// TwinCAT 3 PLC project PlcHammer
// Title: PlcHammer
// Company: Vortex.Library
// ProjectVersion: 0.6.0.913
// ProgramVersion: 3.1.4023.0
// libraries:
//   Tc2_Math, * (Beckhoff Automation GmbH)
//   Tc2_Standard, * (Beckhoff Automation GmbH)
//   Tc2_System, * (Beckhoff Automation GmbH)
//   Tc3_Module, * (Beckhoff Automation GmbH)
//   TcoCore, 0.6.0.913 (Vortex.Library)
//   TcoData, 0.6.0.913 (Vortex.Library)
//   TcoDrivesBeckhoff, 0.6.0.913 (Vortex.Library)
//   TcoElements, 0.6.0.913 (Vortex.Library)
//   TcoInspectors, 0.6.0.913 (Vortex.Library)
//   TcoIo, 0.6.0.913 (Vortex.Library)
//   TcoPneumatics, 0.6.0.913 (Vortex.Library)
//   TcoUtilities, 0.6.0.913 (Vortex.Library)
// project tree:
//   Components/Drive/ DriveSim.TcPOU, DriveSimMoveAbsoluteTask.TcPOU, IDrive.TcIO
//   DUTs/ enumModes.TcDUT
//   Misc/Checkers/ Checkers.TcPOU, AnalogueValueCheck.TcDUT, eCheckResult.TcDUT
//   / PlcTask.TcTTO
//   POUs/ AppContext.TcPOU, TECH_MAIN.TcPOU
//   POUs/Data/ ProcessDataManager.TcPOU, RealValueSimulation.TcPOU, TechnologicalDataManager.TcPOU
//   POUs/Station001/ Station001_Swift.TcPOU, IO.TcGVL, Station001.TcPOU, Station001_Components.TcPOU, Station001_GroundMode.TcPOU, Station001_AutomatMode.TcPOU, Station001_ProductionData.TcDUT, Station001_TechnologicalSettings.TcDUT
// real-time tasks:
//   TASK PlcTask: cycle T#10ms, priority 20, ADS port 350
// motion (NC):
//   TASK NC-Task 1 SAF: cycle T#2ms, priority 4, ADS port 501
//   TASK NC-Task 1 SVB: cycle T#10ms, priority 8, ADS port 511
//   AXIS Axis 1 (id 1)
//     OtherSettings: AllowMotionCmdToSlave=true
//     encoder EncType=1
//     drive DrvType=5
//       Analog: TorqueSetpointScale=10, ScaleFactorActTorque=0.1
//       TimeComp: TaskDelayCycles=1
//     controller CtrType=1
//       CtrPara: PriorControlFactor=1
//         Observer: BandWidth=20
// variable links:
//   PlcHammer/PlcHammer Instance <-> NC-Task 1 SAF/Axes/Axis 1
//     PlcTask Inputs/IO.Axis1.NcToPlc <-> Outputs/ToPlc
//     PlcTask Outputs/IO.Axis1.PlcToNc <-> Inputs/FromPlc

CONFIGURATION PlcHammer
    RESOURCE PLC ON TwinCAT3
        TASK PlcTask(INTERVAL := T#10ms, PRIORITY := 20);
        PROGRAM TECH_MAIN WITH PlcTask : TECH_MAIN;
    END_RESOURCE
END_CONFIGURATION

// ---- DUTs/enumModes.TcDUT
{attribute 'qualified_only'}
{attribute 'strict'}
TYPE enumModes :
(
    Idle := 0,
    Automat := 1000,
    Ground := 2000,
    Service := 3000
);
END_TYPE

// ---- Misc/Checkers/AnalogueValueCheck.TcDUT
{attribute wpf [Container(Layout.Wrap)]}
{attribute wpf [Group(Layout.GroupBox)]}
TYPE AnalogueValueCheck :
STRUCT
    Mininum : REAL;
    {attribute clr [RenderIgnore("ShadowControl", "ShadowControlSlim")]}
    Measured : REAL;
    Maximum : REAL;
END_STRUCT
END_TYPE

// ---- Misc/Checkers/eCheckResult.TcDUT
{attribute 'qualified_only'}
{attribute 'strict'}
TYPE eCheckResult :
(
    None := 0,
    Passed := 10,
    Failed := 20
);
END_TYPE

// ---- POUs/Station001/Station001_ProductionData.TcDUT
TYPE Station001_ProductionData EXTENDS TcoData.TcoEntity :
STRUCT
    {attribute clr [Container(Layout.Stack)]}
    Result : TcoComprehensiveResult;
    RecipeName : STRING;
    DimX : TcoInspectors.TcoAnalogueInspector(THISSTRUCT);
    DimY : TcoInspectors.TcoAnalogueInspector(THISSTRUCT);
    DimZ : TcoInspectors.TcoAnalogueInspector(THISSTRUCT);
END_STRUCT
END_TYPE

// ---- POUs/Station001/Station001_TechnologicalSettings.TcDUT
TYPE Station001_TechnologicalSettings EXTENDS TcoData.TcoEntity :
STRUCT
    LoadPartsHorizontalPosition : LREAL;
    PassedPartsHorizontalPosition : LREAL;
    FailedPartsHorizontalPosition : LREAL;
    AxisSpeed : LREAL;
    AxisAcc : LREAL;
    AxisDcc : LREAL;
    AxisJerk : LREAL;
END_STRUCT
END_TYPE

// ---- POUs/Station001/IO.TcGVL
{attribute 'qualified_only'}
VAR_GLOBAL
    iA1 AT %I* : ARRAY[0..7] OF BOOL;
    iA2 AT %I* : ARRAY[0..7] OF BOOL;
    qA1 AT %Q* : ARRAY[0..7] OF BOOL;
    qA2 AT %Q* : ARRAY[0..7] OF BOOL;
    Axis1 : TcoDrivesBeckhoff.TcoAxisRef;
END_VAR

// ---- Components/Drive/IDrive.TcIO
INTERFACE IDrive

METHOD MoveAbsolute : TcoCore.ITcoTaskStatus
VAR_INPUT
	TargetPosition : LREAL;
END_VAR
END_METHOD

PROPERTY MoveAbsoluteTask : REFERENCE TO DriveSimMoveAbsoluteTask
GET
END_GET
END_PROPERTY

END_INTERFACE

// ---- POUs/TECH_MAIN.TcPOU
PROGRAM TECH_MAIN
VAR
    _app : AppContext;
END_VAR

_app.Run();
_app.RtcSynchronize(TRUE, '', 60);

END_PROGRAM

// ---- POUs/AppContext.TcPOU
FUNCTION_BLOCK AppContext EXTENDS TcoCore.TcoContext
VAR
    _station001 : Station001(THIS^);
END_VAR

(*~
    <docu>
        <summary>
            Main method of the TcoContext. This is the entry point of any control logic that belongs to this context.
            The call of this method is ensured by calling the <c>InstanceName.Run()</c> method, and it must not be called explicitly.
            This method is abstract, and it must be overridden in derived block.
        </summary>
    </docu>
~*)
METHOD PROTECTED Main
THIS^.RtcSynchronize(TRUE, '', 60);
_station001();
END_METHOD

END_FUNCTION_BLOCK

// ---- POUs/Station001/Station001.TcPOU
FUNCTION_BLOCK Station001 EXTENDS TcoCore.TcoObject
VAR
    _components : Station001_Components(THIS^);
    _groundMode : Station001_GroundMode(THIS^, eRestoreMode.None);
    _automatMode : Station001_AutomatMode(THIS^, eRestoreMode.None);
    _swiftSequence : Station001_Swift(THIS^, eRestoreMode.None);
    _groundModeTask : TcoCore.TcoTask(THIS^);
    _automatModeTask : TcoCore.TcoTask(THIS^);
    _serviceModeTask : TcoCore.TcoTask(THIS^);
    _swiftModeTask : TcoCore.TcoTask(THIS^);
    _processRecipies : ProcessDataManager(THIS^);
    _processTraceabilty : ProcessDataManager(THIS^);
    _technologicalDataManager : TechnologicalDataManager(THIS^);
    _currentMode : enumModes := enumModes.Idle;
    _checkers : Checkers(THIS^);
    _externalToken : STRING;
    _externalTokenPresence : BOOL;
END_VAR

_components();
_processRecipies();
_processTraceabilty();
_technologicalDataManager();
ServiceMode();
GroundMode();
AutomatMode();

IF (_swiftModeTask.Execute()) THEN
    Messenger.Trace('Service mode active');
    _automatModeTask.Restore();
    _groundModeTask.Restore();
    _groundMode.Restore();
    _automatMode.Restore();
    _serviceModeTask.Restore();
    _swiftSequence.Run();
    _currentMode := enumModes.Idle;
END_IF

METHOD AutomatMode : BOOL
VAR_INPUT
END_VAR
_automatModeTask.Enabled := _groundModeTask.Done;

IF (_automatModeTask.Execute()) THEN
    Messenger.Trace('Automat mode active');
    _serviceModeTask.Abort();
    _automatMode.Run();
    _currentMode := enumModes.Automat;
END_IF
END_METHOD

PROPERTY Checkers : REFERENCE TO Checkers
GET
Checkers REF= _checkers;
END_GET
END_PROPERTY

PROPERTY Components : REFERENCE TO Station001_Components
GET
Components REF= _components;
END_GET
END_PROPERTY

METHOD GroundMode : BOOL
VAR_INPUT
END_VAR
IF (_groundModeTask.Execute()) THEN
    Messenger.Trace('Ground position mode active');
    _serviceModeTask.Restore();
    _automatModeTask.Restore();
    _automatMode.Restore();
    _groundMode.Run();
    _groundModeTask.DoneWhen(_groundMode.CurrentStep.ID = 300);

    IF _groundModeTask.Done THEN
        _groundMode.Restore();
    END_IF

    _currentMode := enumModes.Ground;
END_IF
END_METHOD

PROPERTY ProcessRecepie : REFERENCE TO ProcessDataManager
GET
ProcessRecepie REF= _processRecipies;
END_GET
END_PROPERTY

PROPERTY ProcessTraceabilty : REFERENCE TO ProcessDataManager
GET
ProcessTraceabilty REF= _processTraceabilty;
END_GET
END_PROPERTY

PROPERTY ProductionData : REFERENCE TO Station001_ProductionData
GET
ProductionData REF= _processTraceabilty._data;
END_GET
END_PROPERTY

METHOD ServiceMode
VAR_INPUT
END_VAR
IF (_serviceModeTask.Execute()) THEN
    Messenger.Trace('Service mode active');
    _automatModeTask.Restore();
    _groundModeTask.Restore();
    _groundMode.Restore();
    _automatMode.Restore();
    _components.Service();
    _currentMode := enumModes.Service;
END_IF
END_METHOD

PROPERTY TechnologicalDataManager : REFERENCE TO TechnologicalDataManager
GET
TechnologicalDataManager REF= _technologicalDataManager;
END_GET
END_PROPERTY

END_FUNCTION_BLOCK

// ---- POUs/Station001/Station001_Components.TcPOU
{attribute wpf [Container(Layout.Stack)]}
FUNCTION_BLOCK Station001_Components EXTENDS TcoCore.TcoObject
VAR
    //	_horizontalAxis : DriveSim(THIS^);
    {attribute addProperty Name "Horizontal axis"}
    _horizontalNcAxis : TcoDrivesBeckhoff.TcoDriveSimple(THIS^);
    {attribute addProperty Name "Vertical piston"}
    {attribute addProperty _moveHomeDefaultName "<#MOVE HOME#>"}
    {attribute addProperty _moveWorkDefaultName "<#MOVE TO WORK#>"}
    {attribute addProperty _stopDefaultName "<#STOP#>"}
    _verticalPiston : TcoPneumatics.TcoCylinder(THIS^);
    {attribute addProperty Name "Gripper piston"}
    {attribute addProperty _moveHomeDefaultName "<#MOVE HOME#>"}
    {attribute addProperty _moveWorkDefaultName "<#MOVE TO WORK#>"}
    {attribute addProperty _stopDefaultName "<#STOP#>"}
    _gripperPiston : TcoPneumatics.TcoCylinder(THIS^);
END_VAR
(* Simulation variables *)
VAR
    _counterSimVerticalPiston : ULINT;
    _counterSimGripperPiston : ULINT;
    _simulationCycleVerticalPiston : BOOL;
    _simulationCycleGripperPiston : BOOL;
    _verticalPosition : INT;
    _gripperPosition : INT;
    _dimXsim : RealValueSimulation;
    _dimYsim : RealValueSimulation;
    _dimZsim : RealValueSimulation;
    _dimX : REAL;
    _dimY : REAL;
    _dimZ : REAL;
END_VAR
VAR CONSTANT
    _verticalPistonStroke : INT := 150;
    _gripperPistonStroke : INT := 50;
END_VAR

Simulation();

_verticalPiston(inoAtHomePos := IO.iA1[0],
    inoAtWorkPos := IO.iA1[1],
    inoToHomePos := IO.qA1[0],
    inoToWorkPos := IO.qA1[1]);

_gripperPiston(inoAtHomePos := IO.iA1[2],
    inoAtWorkPos := IO.iA1[3],
    inoToHomePos := IO.qA1[2],
    inoToWorkPos := IO.qA1[3]);

//_horizontalAxis();
_horizontalNcAxis(inEnable := TRUE,
    inEnablePositive := TRUE,
    inEnableNegative := TRUE,
    inCalibrationCam := FALSE,
    inoAxisRef := IO.Axis1);

PROPERTY Gripper : REFERENCE TO TcoPneumatics.TcoCylinder
GET
Gripper REF= _gripperPiston;
END_GET
END_PROPERTY

PROPERTY HorizontalNcAxis : TcoDrivesBeckhoff.ITcoDriveSimple
GET
HorizontalNcAxis := _horizontalNcAxis;
END_GET
END_PROPERTY

METHOD Service : BOOL
VAR_INPUT
END_VAR
//_horizontalAxis.Service();
_horizontalNcAxis.Service();
_verticalPiston.Service();
_gripperPiston.Service();
END_METHOD

METHOD Simulation
VAR_INPUT
END_VAR
IF (_verticalPiston.MoveHomeTask.Busy OR _verticalPiston.MoveWorkTask.Busy) THEN
    _counterSimVerticalPiston := _counterSimVerticalPiston + 1;
    _simulationCycleVerticalPiston := (_counterSimVerticalPiston MOD _verticalPistonStroke) = 0;
END_IF;

IF (Gripper.MoveHomeTask.Busy OR Gripper.MoveWorkTask.Busy) THEN
    _counterSimGripperPiston := _counterSimVerticalPiston + 1;
    _simulationCycleGripperPiston := (_counterSimVerticalPiston MOD _gripperPistonStroke) = 0;
END_IF;

IF (IO.qA1[0] AND _simulationCycleVerticalPiston) THEN
    IO.iA1[0] := TRUE;
    IO.iA1[1] := FALSE;
    _verticalPosition := 0;
END_IF

IF (IO.qA1[1] AND _simulationCycleVerticalPiston) THEN
    IO.iA1[1] := TRUE;
    IO.iA1[0] := FALSE;
    _verticalPosition := _verticalPistonStroke;
END_IF

IF (IO.qA1[0] AND NOT IO.iA1[0]) THEN
    _verticalPosition := (_verticalPosition - 1);
END_IF;

IF (IO.qA1[1] AND NOT IO.iA1[1]) THEN
    _verticalPosition := (_verticalPosition + 1);
END_IF;

IF (IO.qA1[2] AND _simulationCycleVerticalPiston) THEN
    IO.iA1[2] := TRUE;
    IO.iA1[3] := FALSE;
    _gripperPosition := 0;
END_IF

IF (IO.qA1[3] AND _simulationCycleVerticalPiston) THEN
    IO.iA1[3] := TRUE;
    IO.iA1[2] := FALSE;
    _gripperPosition := _gripperPistonStroke;
END_IF

IF (IO.qA1[2] AND NOT IO.iA1[2]) THEN
    _gripperPosition := (_gripperPosition - 1);
END_IF;

IF (IO.qA1[3] AND NOT IO.iA1[3]) THEN
    _gripperPosition := (_gripperPosition + 1);
END_IF

_dimXsim.Dc := 3;
_dimYsim.Dc := 3;
_dimZsim.Dc := 3;
_dimXsim.P1 := 0.74;
_dimYsim.P1 := 0.74;
_dimZsim.P1 := 0.74;
_dimXsim.P2 := 1.1;
_dimYsim.P2 := 1.1;
_dimZsim.P2 := 1.1;
END_METHOD

PROPERTY VerticalAxis : REFERENCE TO TcoPneumatics.TcoCylinder
GET
VerticalAxis REF= _verticalPiston;
END_GET
END_PROPERTY

END_FUNCTION_BLOCK

// ---- POUs/Data/RealValueSimulation.TcPOU
FUNCTION_BLOCK RealValueSimulation
VAR_INPUT
    inMinValue : REAL;
    inMaxValue : REAL;
END_VAR
VAR_IN_OUT
    inoutValue : REAL;
END_VAR
VAR
    _dc : LREAL := 5.4;
    _min : REAL;
    _max : REAL;
    _p1 : LREAL := 2;
    _p2 : LREAL := 3.5;
    _x0 : LREAL;
    _x1 : LREAL;
    _pm : LREAL;
    _ex : LREAL;
END_VAR

_ex := EXPT(10, _dc);
_x0 := inoutValue * _ex;

IF _x0 = 0 THEN
    _x0 := (inMaxValue + inMinValue) / 2 * _ex;
END_IF

_min := inMinValue * _ex;
_max := inMaxValue * _ex;
_pm := (_max - _min);
_x1 := _min + (Tc2_Math.LMOD((_x0 * _p1 + _p2), _pm));
inoutValue := Tc2_Math.LTRUNC(_x1 / _ex);

PROPERTY Dc : LREAL
GET
Dc := _dc;
END_GET
SET
_dc := Dc;
END_SET
END_PROPERTY

PROPERTY P1 : LREAL
GET
P1 := _p1;
END_GET
SET
_p1 := P1;
END_SET
END_PROPERTY

PROPERTY P2 : LREAL
GET
P2 := _p2;
END_GET
SET
_p2 := P2;
END_SET
END_PROPERTY

END_FUNCTION_BLOCK

// ---- POUs/Station001/Station001_GroundMode.TcPOU
FUNCTION_BLOCK Station001_GroundMode EXTENDS TcoCore.TcoSequencer

(*~
    <docu>
        <summary>
            Main method of the sequener. Custom code needs to be placed here. The sequencer is executed by call of InstanceName.Run() method.
            This method is abstract, and it must be overridden in derived block.
        </summary>
    </docu>
~*)
METHOD PROTECTED Main : BOOL
VAR CONSTANT
    HORIZONTAL_AXIS_HOME_POSITION : LREAL := 0.0;
END_VAR
IF (Step(10, TRUE, 'RESTORE ALL COMPONENTS')) THEN
    //--------------------------------------------
    Station.Components._horizontalNcAxis.Restore();
    Station.Components._verticalPiston.Restore();
    Station.Components._gripperPiston.Restore();
    StepCompleteWhen(TRUE);
    //--------------------------------------------
END_IF;

IF (Step(100, TRUE, 'MOVE VERTICAL AXIS UP')) THEN
    //--------------------------------------------
    StepCompleteWhen(Station.Components.VerticalAxis.MoveToHome().Done);
    //--------------------------------------------
END_IF;

IF (Step(125, TRUE, 'LOAD TECHNOLOGICAL SETTINGS')) THEN
    //--------------------------------------------
    StepCompleteWhen(Station.TechnologicalDataManager.Read('default').Done);
    //--------------------------------------------
END_IF;

IF (Step(150, NOT Station.Components.HorizontalNcAxis.DriveRef._axisStatus.Homed, 'HORIZONTAL AXIS HOMING')) THEN
    //--------------------------------------------
    StepCompleteWhen(Station.Components.HorizontalNcAxis.DriveRef.Home(inPosition := 0,
            inHomingMode := TcoDrivesBeckhoff.eHomingMode.MC_Direct,
            inClearPositionLag := FALSE,
            inSearchDirection := TcoDrivesBeckhoff.eDirection.MC_Undefined_Direction,
            inSearchVelocity := 100.0,
            inSyncDirection := TcoDrivesBeckhoff.eDirection.MC_Undefined_Direction,
            inSyncVelocity := 100.0,
            inReferenceMode := TcoDrivesBeckhoff.eEncoderReferenceMode.ENCODERREFERENCEMODE_DEFAULT).Done);
    //--------------------------------------------
END_IF;

IF (Step(200, TRUE, 'MOVE HORIZONTAL AXIS TO BASE POSITION & OPEN GRIPPER')) THEN
    //--------------------------------------------
    IF (Station.Components.HorizontalNcAxis.DriveRef.MoveAbsolute(HORIZONTAL_AXIS_HOME_POSITION,
        THIS^.Station.TechnologicalDataManager._data.AxisSpeed,
        THIS^.Station.TechnologicalDataManager._data.AxisAcc,
        THIS^.Station.TechnologicalDataManager._data.AxisDcc,
        THIS^.Station.TechnologicalDataManager._data.AxisJerk).Done AND
        Station.Components.Gripper.MoveToHome().Done) THEN
        CompleteStep();
    END_IF;
    //--------------------------------------------
END_IF;

IF (Step(300, TRUE, 'GROUND POSITION DONE')) THEN
    //--------------------------------------------
    ;
    //--------------------------------------------
END_IF;
END_METHOD

(*~
    <docu>
        <summary>
            This method is executed upon step completion.
            This method can be overridden in derived block by custom logic.
        </summary>
    </docu>
~*)
METHOD PROTECTED OnStepCompleted
END_METHOD

PROPERTY Station : REFERENCE TO Station001
GET
VAR
    _station : POINTER TO Station001;
END_VAR
IF __QUERYPOINTER(Parent, _station) THEN // Check if _Parent is Station001
    Station REF= _station^; // If the check is successful dereference a pointer. simlar to THIS^ or SUPER^
END_IF
END_GET
END_PROPERTY

END_FUNCTION_BLOCK

// ---- POUs/Data/TechnologicalDataManager.TcPOU
FUNCTION_BLOCK TechnologicalDataManager EXTENDS TcoData.TcoDataExchange
VAR
    //this variable has to called "_data" - PC app will access this variable by its name.
    _data : Station001_TechnologicalSettings := (Parent := THIS^);
END_VAR

SUPER^();
//Set som default values in case of no setting loaded to the PLC yet.
//IF _data.LoadPartsHorizontalPosition = 0  AND _data.FailedPartsHorizontalPosition = 0 AND _data.PassedPartsHorizontalPosition = 0 THEN
//    _data.LoadPartsHorizontalPosition := 50;
//    _data.FailedPartsHorizontalPosition := 300.0;
//    _data.PassedPartsHorizontalPosition := 450.0;
//END_IF
//IF _data.AxisSpeed = 0 THEN
//    _data.AxisSpeed := 1000.0;
//END_IF
//IF _data.AxisAcc = 0 THEN
//    _data.AxisAcc := 10000.0;
//END_IF
//IF _data.AxisDcc = 0 THEN
//    _data.AxisDcc := 10000.0;
//END_IF
//IF _data.AxisJerk = 0 THEN
//    _data.AxisJerk := 50000.0;
//END_IF

END_FUNCTION_BLOCK

// ---- POUs/Station001/Station001_AutomatMode.TcPOU
FUNCTION_BLOCK Station001_AutomatMode EXTENDS TcoCore.TcoSequencer
VAR
    _partPassedChecks : BOOL;
    _groupInspection : TcoInspectors.TcoInspectionGroup(THIS^);
    _dialog : TcoCore.TcoDialog(THIS^);
END_VAR

(*~
    <docu>
        <summary>
            Main method of the sequener. Custom code needs to be placed here. The sequencer is executed by call of InstanceName.Run() method.
            This method is abstract, and it must be overridden in derived block.
        </summary>
    </docu>
~*)
METHOD PROTECTED Main : BOOL
VAR CONSTANT
    HORIZONTAL_AXIS_HOME_POSITION : LREAL := 100.0;
END_VAR
VAR_INST
    _id : STRING;
END_VAR
IF (Step(0, TRUE, 'DIALOG - DO WE CONTINUE')) THEN
    //--------------------------------------------
    IF (_dialog.Show().WithOk().WithCaption('What`s next?').WithText('To continue click OK?').Answer = TcoCore.eDialogAnswer.OK) THEN
        CompleteStep();
    END_IF;
    //--------------------------------------------
END_IF;

IF (Step(10, TRUE, 'MOVE HORIZONTAL TO LOAD')) THEN
    //--------------------------------------------
    StepCompleteWhen(Station.Components.HorizontalNCAxis.DriveRef
            .MoveAbsolute(THIS^.Station.TechnologicalDataManager._data.LoadPartsHorizontalPosition,
                THIS^.Station.TechnologicalDataManager._data.AxisSpeed,
                THIS^.Station.TechnologicalDataManager._data.AxisAcc,
                THIS^.Station.TechnologicalDataManager._data.AxisDcc,
                THIS^.Station.TechnologicalDataManager._data.AxisJerk).Done);
    //--------------------------------------------
END_IF;

IF (Step(25, TRUE, 'LOAD TECHNOLOGICAL SETTINGS')) THEN
    //--------------------------------------------
    IF (NOT Station.TechnologicalDataManager.Messenger.OnCondition(Station.TechnologicalDataManager._data._EntityId = '')
        .Error('Technological settings not selected.')
        .Pin().Pinned) THEN
        ;
        StepCompleteWhen(Station.TechnologicalDataManager.Read(Identifier := Station.TechnologicalDataManager._data._EntityId).Done);
    END_IF;
    //--------------------------------------------
END_IF;

IF (Step(50, TRUE, 'LOAD RECIPE SETTINGS')) THEN
    //--------------------------------------------
    IF (NOT Station.ProcessRecepie.Messenger.OnCondition(Station.ProcessRecepie._data._EntityId = '').Error('Process settings not selected.').Pin()
        .Pinned) THEN
        StepCompleteWhen(Station.ProcessRecepie.Read(Identifier := Station.ProcessRecepie._data._EntityId).Done);
        Station.ProductionData := Station.ProcessRecepie._data;
    END_IF

    //--------------------------------------------
END_IF;

IF (Step(100, TRUE, 'MOVE VERTICAL AXIS DOWN')) THEN
    //--------------------------------------------
    StepCompleteWhen(Station.Components.VerticalAxis.MoveToWork().Done);
    //--------------------------------------------
END_IF;

IF (Step(150, TRUE, 'GENERATE SIMULATED VALUES')) THEN
    //--------------------------------------------
    Station.Components._dimXsim(inMinValue := Station.ProductionData.DimX.Data.RequiredMin + 50,
        inMaxValue := Station.ProductionData.DimX.Data.RequiredMax - 50,
        inoutValue := Station.Components._dimX);

    Station.Components._dimYsim(inMinValue := Station.ProductionData.DimY.Data.RequiredMin + 50,
        inMaxValue := Station.ProductionData.DimY.Data.RequiredMax - 50,
        inoutValue := Station.Components._dimY);

    Station.Components._dimZsim(inMinValue := Station.ProductionData.DimZ.Data.RequiredMin + 50,
        inMaxValue := Station.ProductionData.DimZ.Data.RequiredMax - 50,
        inoutValue := Station.Components._dimZ);

    StepCompleteWhen(TRUE);
    //--------------------------------------------
END_IF;

IF (Step(200, TRUE, 'CHECK DIMENSIONS')) THEN
    //--------------------------------------------
    _groupInspection.WithCoordinator(THIS^)
        .Act()
        .Inspect(Station.ProcessTraceabilty._data.DimX.Inspect(Station.Components._dimX))
        .Inspect(Station.ProcessTraceabilty._data.DimY.Inspect(Station.Components._dimY))
        .Inspect(Station.ProcessTraceabilty._data.DimZ.Inspect(Station.Components._dimZ))
        .UpdateComprehensiveResult(Station.ProcessTraceabilty._data.Result)
        .OnFail().Dialog(200);
    //--------------------------------------------
END_IF;

IF (Step(300, TRUE, 'CLOSE GRIPPER')) THEN
    //--------------------------------------------
    StepCompleteWhen(Station.Components.Gripper.MoveToWork().Done);
    //--------------------------------------------
END_IF;

IF (Step(400, TRUE, 'MOVE VERTICAL AXIS UP')) THEN
    //--------------------------------------------
    StepCompleteWhen(Station.Components.VerticalAxis.MoveToHome().Done);
    //--------------------------------------------
END_IF;

IF (Step(425, _partPassedChecks, 'MOVE HORIZONTAL AXIS TO UNLOAD POSITION (PASSED CONVEYOR)')) THEN
    //--------------------------------------------
    StepCompleteWhen(Station.Components.HorizontalNcAxis.DriveRef
            .MoveAbsolute(THIS^.Station.TechnologicalDataManager._data.PassedPartsHorizontalPosition,
                THIS^.Station.TechnologicalDataManager._data.AxisSpeed,
                THIS^.Station.TechnologicalDataManager._data.AxisAcc,
                THIS^.Station.TechnologicalDataManager._data.AxisDcc,
                THIS^.Station.TechnologicalDataManager._data.AxisJerk).Done);
    //--------------------------------------------
END_IF;

IF (Step(450, NOT _partPassedChecks, 'MOVE HORIZONTAL AXIS TO UNLOAD POSITION (FAILED CONVEYOR)')) THEN
    //--------------------------------------------
    StepCompleteWhen(Station.Components.HorizontalNcAxis.DriveRef
            .MoveAbsolute(THIS^.Station.TechnologicalDataManager._data.FailedPartsHorizontalPosition,
                THIS^.Station.TechnologicalDataManager._data.AxisSpeed,
                THIS^.Station.TechnologicalDataManager._data.AxisAcc,
                THIS^.Station.TechnologicalDataManager._data.AxisDcc,
                THIS^.Station.TechnologicalDataManager._data.AxisJerk).Done);
    //--------------------------------------------
END_IF;

IF (Step(500, TRUE, 'MOVE VERTICAL AXIS TO UNLOAD POSITION')) THEN
    //--------------------------------------------
    StepCompleteWhen(Station.Components.VerticalAxis.MoveToWork().Done);
    //--------------------------------------------
END_IF;

IF (Step(600, TRUE, 'OPEN GRIPPER')) THEN
    //--------------------------------------------
    StepCompleteWhen(Station.Components.Gripper.MoveToHome().Done);
    //--------------------------------------------
END_IF;

IF (Step(700, TRUE, 'MOVE VERTICAL UP')) THEN
    //--------------------------------------------
    StepCompleteWhen(Station.Components.VerticalAxis.MoveToHome().Done);
    //--------------------------------------------
END_IF;

IF (Step(800, TRUE, 'MOVE HORIZONTAL TO LOAD - ASYNC')) THEN
    //--------------------------------------------
    Station.Components.HorizontalNCAxis.DriveRef.MoveAbsolute(THIS^.Station.TechnologicalDataManager._data.LoadPartsHorizontalPosition,
        THIS^.Station.TechnologicalDataManager._data.AxisSpeed,
        THIS^.Station.TechnologicalDataManager._data.AxisAcc,
        THIS^.Station.TechnologicalDataManager._data.AxisDcc,
        THIS^.Station.TechnologicalDataManager._data.AxisJerk);

    StepCompleteWhen(TRUE);
    //--------------------------------------------
END_IF;

IF (Step(840, TRUE, 'CHECK THAT THE HORIZONTAL AXIS IS IN POSITION')) THEN
    //--------------------------------------------
    _id := ULINT_TO_STRING(THIS^.Context.RealTimeClock.TickClock());
    StepCompleteWhen(TRUE);
    //--------------------------------------------
END_IF;

IF (Step(850, TRUE, 'SAVE DATA')) THEN
    //--------------------------------------------
    StepCompleteWhen(Station.ProcessTraceabilty.Create(Identifier := _id).Done);
    //--------------------------------------------
END_IF;

IF (Step(900, TRUE, 'CHECK THAT THE HORIZONTAL AXIS IS IN POSITION')) THEN
    //--------------------------------------------
    StepCompleteWhen(Station.Components.HorizontalNcAxis.DriveRef.MoveAbsoluteTask.Done);
    //--------------------------------------------
END_IF;

IF (Step(THIS^.RESTORE_STEP_ID, TRUE, 'MOVE VERTICAL AXIS UP')) THEN
    //--------------------------------------------
    StepCompleteWhen(Station.Components.VerticalAxis.MoveToHome().Done);
    //--------------------------------------------
END_IF;

IF (Step(37000, TRUE, 'MOVE HORIZONTAL AXIS TO BASE POSITION & OPEN GRIPPER')) THEN
    //--------------------------------------------
    IF (Station.Components.HorizontalNcAxis.DriveRef.MoveAbsolute(THIS^.Station.TechnologicalDataManager._data.LoadPartsHorizontalPosition,
        THIS^.Station.TechnologicalDataManager._data.AxisSpeed,
        THIS^.Station.TechnologicalDataManager._data.AxisAcc,
        THIS^.Station.TechnologicalDataManager._data.AxisDcc,
        THIS^.Station.TechnologicalDataManager._data.AxisJerk).Done AND
        Station.Components.Gripper.MoveToHome().Done) THEN
        CompleteStep();
    END_IF;
    //--------------------------------------------
END_IF;

IF (Step(1000, TRUE, 'SEUQNCE COMPLETE')) THEN
    //--------------------------------------------
    CompleteSequence();
    //--------------------------------------------
END_IF;
END_METHOD

(*~
    <docu>
        <summary>
            This method is executed upon step completion.
            This method can be overridden in derived block by custom logic.
        </summary>
    </docu>
~*)
METHOD PROTECTED OnStepCompleted
END_METHOD

PROPERTY Station : REFERENCE TO Station001
GET
VAR
    _station : POINTER TO Station001;
END_VAR
IF __QUERYPOINTER(Parent, _station) THEN // Check if _Parent is Station001
    Station REF= _station^; // If the check is successful dereference a pointer. simlar to THIS^ or SUPER^
END_IF
END_GET
END_PROPERTY

END_FUNCTION_BLOCK

// ---- POUs/Station001/Station001_Swift.TcPOU
FUNCTION_BLOCK Station001_Swift EXTENDS TcoCore.TcoSequencer
VAR
    _partPassedChecks : BOOL;
END_VAR

(*~
    <docu>
        <summary>
            Main method of the sequener. Custom code needs to be placed here. The sequencer is executed by call of InstanceName.Run() method.
            This method is abstract, and it must be overridden in derived block.
        </summary>
    </docu>
~*)
METHOD PROTECTED Main : BOOL
VAR CONSTANT
    HORIZONTAL_AXIS_HOME_POSITION : LREAL := 100.0;
END_VAR
IF Step(10, TRUE, 'TECH_MAIN._app._station001._components._gripperPiston._moveHomeDefault') THEN
    //-------------------------------------------------------
    IF (TECH_MAIN._app._station001._components._gripperPiston._moveHomeDefault.Invoke().Done) THEN
        StepCompleteWhen(TRUE);
    END_IF;
    //-------------------------------------------------------
END_IF;

IF Step(20, TRUE, 'TECH_MAIN._app._station001._components._verticalPiston._moveHomeDefault') THEN
    //-------------------------------------------------------
    IF (TECH_MAIN._app._station001._components._verticalPiston._moveHomeDefault.Invoke().Done) THEN
        StepCompleteWhen(TRUE);
    END_IF;
    //-------------------------------------------------------
END_IF;

IF Step(30, TRUE, 'TECH_MAIN._app._station001._components._horizontalNcAxis') THEN
    //-------------------------------------------------------
    IF (TECH_MAIN._app._station001._components._horizontalNcAxis.MoveAbsolute(inPosition := 450,
        inVelocity := 1000,
        inAcceleration := 10000,
        inDeceleration := 10000,
        inJerk := 50000).Done) THEN
        StepCompleteWhen(TRUE);
    END_IF;
    //-------------------------------------------------------
END_IF;

IF Step(40, TRUE, 'TECH_MAIN._app._station001._components._verticalPiston._moveWorkDefault') THEN
    //-------------------------------------------------------
    IF (TECH_MAIN._app._station001._components._verticalPiston._moveWorkDefault.Invoke().Done) THEN
        StepCompleteWhen(TRUE);
    END_IF;
    //-------------------------------------------------------
END_IF;

IF Step(50, TRUE, 'TECH_MAIN._app._station001._components._gripperPiston._moveWorkDefault') THEN
    //-------------------------------------------------------
    IF (TECH_MAIN._app._station001._components._gripperPiston._moveWorkDefault.Invoke().Done) THEN
        StepCompleteWhen(TRUE);
    END_IF;
    //-------------------------------------------------------
END_IF;

IF Step(60, TRUE, 'TECH_MAIN._app._station001._components._gripperPiston._moveHomeDefault') THEN
    //-------------------------------------------------------
    IF (TECH_MAIN._app._station001._components._gripperPiston._moveHomeDefault.Invoke().Done) THEN
        StepCompleteWhen(TRUE);
    END_IF;
    //-------------------------------------------------------
END_IF;

IF Step(70, TRUE, 'TECH_MAIN._app._station001._components._verticalPiston._moveHomeDefault') THEN
    //-------------------------------------------------------
    IF (TECH_MAIN._app._station001._components._verticalPiston._moveHomeDefault.Invoke().Done) THEN
        StepCompleteWhen(TRUE);
    END_IF;
    //-------------------------------------------------------
END_IF;

IF Step(80, TRUE, 'TECH_MAIN._app._station001._components._horizontalNcAxis') THEN
    //-------------------------------------------------------
    IF (TECH_MAIN._app._station001._components._horizontalNcAxis.MoveAbsolute(inPosition := 0,
        inVelocity := 1000,
        inAcceleration := 10000,
        inDeceleration := 10000,
        inJerk := 50000).Done) THEN
        StepCompleteWhen(TRUE);
    END_IF;
    //-------------------------------------------------------
END_IF;

IF Step(90, TRUE, 'TECH_MAIN._app._station001._components._verticalPiston._moveWorkDefault') THEN
    //-------------------------------------------------------
    IF (TECH_MAIN._app._station001._components._verticalPiston._moveWorkDefault.Invoke().Done) THEN
        StepCompleteWhen(TRUE);
    END_IF;
    //-------------------------------------------------------
END_IF;

IF Step(100, TRUE, 'TECH_MAIN._app._station001._components._gripperPiston._moveWorkDefault') THEN
    //-------------------------------------------------------
    IF (TECH_MAIN._app._station001._components._gripperPiston._moveWorkDefault.Invoke().Done) THEN
        StepCompleteWhen(TRUE);
    END_IF;
    //-------------------------------------------------------
END_IF;

IF Step(110, TRUE, 'TECH_MAIN._app._station001._components._horizontalNcAxis') THEN
    //-------------------------------------------------------
    IF (TECH_MAIN._app._station001._components._horizontalNcAxis.MoveAbsolute(inPosition := 200,
        inVelocity := 1000,
        inAcceleration := 10000,
        inDeceleration := 10000,
        inJerk := 50000).Done) THEN
        StepCompleteWhen(TRUE);
    END_IF;
    //-------------------------------------------------------
END_IF;
END_METHOD

(*~
    <docu>
        <summary>
            This method is executed upon step completion.
            This method can be overridden in derived block by custom logic.
        </summary>
    </docu>
~*)
METHOD PROTECTED OnStepCompleted
END_METHOD

PROPERTY Station : REFERENCE TO Station001
GET
VAR
    _station : POINTER TO Station001;
END_VAR
IF __QUERYPOINTER(Parent, _station) THEN // Check if _Parent is Station001
    Station REF= _station^; // If the check is successful dereference a pointer. simlar to THIS^ or SUPER^
END_IF
END_GET
END_PROPERTY

END_FUNCTION_BLOCK

// ---- POUs/Data/ProcessDataManager.TcPOU
FUNCTION_BLOCK ProcessDataManager EXTENDS TcoData.TcoDataExchange
VAR
    //this variable has to called "_data" - PC app will access this variable by its name.
    {attribute clr [Container(Layout.Tabs)]}
    {attribute clr [Group(Layout.Scroll)]}
    _data : Station001_ProductionData := (Parent := THIS^);
END_VAR

SUPER^();
//Set default values in case that no setting has been loaded into the PLC yet.
//IF _data.DimX.Mininum = 0 AND _data.DimX.Maximum = 0 THEN
//    _data.DimX.Mininum :=
//        0.95 * MAIN._app._station001._components._dimXsim.inMinValue + 0.05 * MAIN._app._station001._components._dimXsim.inMaxValue;
//    _data.DimX.Maximum :=
//        0.05 * MAIN._app._station001._components._dimXsim.inMinValue + 0.95 * MAIN._app._station001._components._dimXsim.inMaxValue;
//END_IF
//IF _data.DimY.Mininum = 0 AND _data.DimY.Maximum = 0 THEN
//    _data.DimY.Mininum :=
//        0.95 * MAIN._app._station001._components._dimYsim.inMinValue + 0.05 * MAIN._app._station001._components._dimYsim.inMaxValue;
//    _data.DimY.Maximum :=
//        0.05 * MAIN._app._station001._components._dimYsim.inMinValue + 0.95 * MAIN._app._station001._components._dimYsim.inMaxValue;
//END_IF
//IF _data.DimZ.Mininum = 0 AND _data.DimZ.Maximum = 0 THEN
//    _data.DimZ.Mininum :=
//        0.95 * MAIN._app._station001._components._dimZsim.inMinValue + 0.05 * MAIN._app._station001._components._dimZsim.inMaxValue;
//    _data.DimZ.Maximum :=
//        0.05 * MAIN._app._station001._components._dimZsim.inMinValue + 0.95 * MAIN._app._station001._components._dimZsim.inMaxValue;
//END_IF

METHOD SetDataResult
VAR_INPUT
    Result : TcoComprehensiveResult;
END_VAR
_data.Result := Result;
END_METHOD

METHOD SetRecipe
VAR_INPUT
    RecipeName : STRING;
END_VAR
_data.RecipeName := RecipeName;
END_METHOD

END_FUNCTION_BLOCK

// ---- Misc/Checkers/Checkers.TcPOU
FUNCTION_BLOCK Checkers EXTENDS TcoCore.TcoObject
VAR
    _result : eCheckResult;
END_VAR

METHOD CheckAnalogue : REFERENCE TO Checkers
VAR_INPUT
    Signal : REAL;
END_VAR
VAR_INPUT
    pData : POINTER TO AnalogueValueCheck;
END_VAR
VAR
    _inRange : BOOL;
END_VAR
pData^.Measured := Signal;
_inRange := (Signal >= pData^.Mininum) AND (Signal <= pData^.Maximum);

IF (NOT _inRange AND_THEN _result <= eCheckResult.Passed) THEN
    _result := eCheckResult.Failed;
END_IF;

CheckAnalogue REF= THIS^;
END_METHOD

METHOD HasPassed : BOOL
VAR_INPUT
END_VAR
HasPassed := _result = eCheckResult.Passed;
_result := eCheckResult.None;
END_METHOD

METHOD StartChecks : REFERENCE TO Checkers
VAR_INPUT
END_VAR
_result := eCheckResult.Passed;
StartChecks REF= THIS^;
END_METHOD

END_FUNCTION_BLOCK

// ---- Components/Drive/DriveSim.TcPOU
FUNCTION_BLOCK DriveSim EXTENDS TcoCore.TcoComponent IMPLEMENTS IDrive
VAR
    {attribute addProperty Name "<#Current position#>"}
    _position : LREAL;
END_VAR
VAR
    {attribute addProperty Name "<#Move absolute#>"}
    {attribute addProperty ToolTip "<#Moves the drive to absolute position given by parameter 'Target Position'#>"}
    _moveAbsoluteTask : DriveSimMoveAbsoluteTask(THIS^);
END_VAR

_moveAbsoluteTask(_drive := THIS^);

METHOD MoveAbsolute : TcoCore.ITcoTaskStatus
VAR_INPUT
    TargetPosition : LREAL;
END_VAR
_moveAbsoluteTask.TargetPosition := TargetPosition;
MoveAbsolute := _moveAbsoluteTask.Invoke();
END_METHOD

PROPERTY MoveAbsoluteTask : REFERENCE TO DriveSimMoveAbsoluteTask
GET
MoveAbsoluteTask REF= _moveAbsoluteTask;
END_GET
END_PROPERTY

PROPERTY Position : LREAL
GET
Position := _position;
END_GET
SET
_position := Position;
END_SET
END_PROPERTY

(*~
    <docu>
        <summary>
            Restores this instance to the Ready state. Can be called explicitly or from within one of the restore mechanisms.
        </summary>
    </docu>
~*)
METHOD Restore : ITcoRestorable
END_METHOD

(*~
    <docu>
        <summary>
            Custom service (manual, maintenance) logic.
            This method must be implemented in derived class.
        </summary>
    </docu>
~*)
METHOD PROTECTED ServiceMode
END_METHOD

END_FUNCTION_BLOCK

// ---- Components/Drive/DriveSimMoveAbsoluteTask.TcPOU
FUNCTION_BLOCK DriveSimMoveAbsoluteTask EXTENDS TcoCore.TcoTask
VAR_IN_OUT
    _drive : DriveSim;
END_VAR
VAR
    {attribute addProperty Name "<#Target position#>"}
    _targetPosition : LREAL;
END_VAR

IF (Execute()) THEN
    Messenger.Debug('Moving absolute');

    IF (_drive.Position < _targetPosition) THEN
        _drive.Position := _drive._position + 1;
    ELSE
        _drive.Position := _drive._position - 1;
    END_IF;

    DoneWhen(ABS(_drive._position - THIS^.TargetPosition) < 2);
END_IF

PROPERTY TargetPosition : LREAL
GET
TargetPosition := _targetPosition;
END_GET
SET
_targetPosition := TargetPosition;
END_SET
END_PROPERTY

END_FUNCTION_BLOCK
